{attribute 'qualified_only'}
VAR_GLOBAL
	StateProteza : UDINT;
	StateCurrentProteza : DINT;
	BoolProteza  :  BOOL := 1 ;
END_VAR

(* stored: Version 1.1.0.1
   GVL GlobalVariableList: Id {e704112c-6181-0958-0436-a320982b8db1} *)
